// TIA Portal V19 export
TYPE "Prg_Pivot"
// stored: Access Published
   STRUCT
      PrgNo : DInt;
      PrgName : String[30];
      RecordNo : Int;   // Record Number: 1..PPRG_TOTAL_ARCHIVE_ITEMS
   END_STRUCT;
END_TYPE
